// Mitsubishi GX Works2 project: ex1   PLC: Q03UDV

PROGRAM MAIN
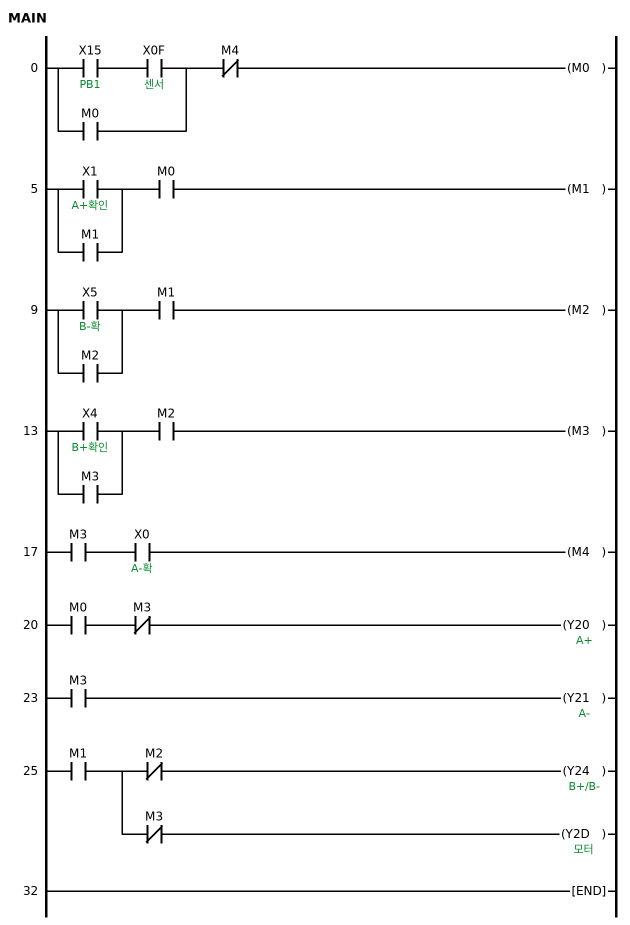
0     LD      X15  ; PB1
      AND     X0F  ; 센서
      OR      M0
      ANI     M4
      OUT     M0
5     LD      X1  ; A+확인
      OR      M1
      AND     M0
      OUT     M1
9     LD      X5  ; B-확
      OR      M2
      AND     M1
      OUT     M2
13    LD      X4  ; B+확인
      OR      M3
      AND     M2
      OUT     M3
17    LD      M3
      AND     X0  ; A-확
      OUT     M4
20    LD      M0
      ANI     M3
      OUT     Y20  ; A+
23    LD      M3
      OUT     Y21  ; A-
25    LD      M1
      MPS
      ANI     M2
      OUT     Y24  ; B+/B-
      MPP
      ANI     M3
      OUT     Y2D  ; 모터
32    END
END_PROGRAM
